// SIMATIC S7-200 SMART project (STEP 7-Micro/WIN SMART), CPU SR20

SYMBOL_TABLE 系统符号
Always_On        SM0.0    // 始终接通
END_SYMBOL_TABLE

ORGANIZATION_BLOCK MAIN:OB1
TITLE=程序注释
BEGIN
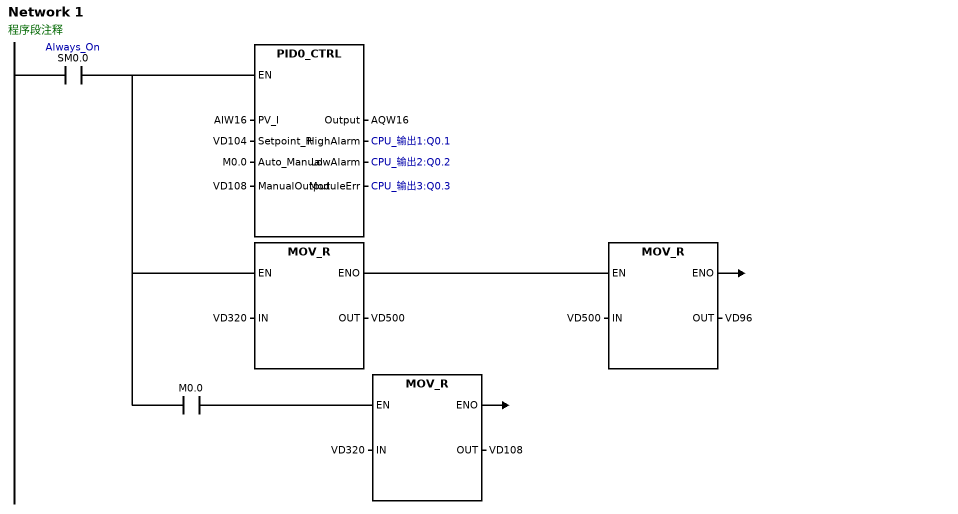
Network 1
// 程序段注释
LD     Always_On:SM0.0
LPS
CALL   PID0_CTRL:SBR0, AIW16, VD104, M0.0, VD108, AQW16, CPU_输出1:Q0.1, CPU_输出2:Q0.2, CPU_输出3:Q0.3
MOVR   VD320, VD500
AENO
MOVR   VD500, VD96
LPP
A      M0.0
MOVR   VD320, VD108
END_ORGANIZATION_BLOCK

// SBR0: protected block, not included

// INT1: protected block, not included
